// TIA Portal V20 export
TYPE "UDT_MTP_StringReportValue"
   STRUCT
      WQC { ExternalWritable := 'False'} : Byte := 16#FF;   // Worst Quality Code
      Text { ExternalWritable := 'False'} : String[40];   // Value
      MissedValue { ExternalWritable := 'False'} : Bool;   // MissedValueFeature
   END_STRUCT;
END_TYPE
